// TIA Portal project "学习计数器" (V15.1)

(* hardware
DEVICE "S7-1200 station_1"  S7-1200 Station
   slot 0: "Rack_0"  S7-1200 Rack  Rack  V1.0
   slot 1: "PLC_1"  CPU 1214C DC/DC/DC  6ES7 214-1AG40-0XB0  V4.2
*)

// ===== PLC "PLC_1"  CPU 1214C DC/DC/DC =====

VAR_GLOBAL   // PLC tag table "默认变量表"
   "Tag_1" AT %M0.0 : Bool;
   "Tag_2" AT %M0.1 : Bool;
   "Tag_3" AT %MW100 : Int;
   "Tag_4" AT %Q0.0 : Bool;
   "Tag_5" AT %Q0.1 : Bool;
   "Tag_6" AT %M0.2 : Bool;
   "Tag_7" AT %M0.3 : Bool;
   "Tag_8" AT %MW101 : Int;
   "Tag_9" AT %M0.4 : Bool;
   "Tag_10" AT %M0.5 : Bool;
   "Tag_11" AT %M0.6 : Bool;
   "Tag_12" AT %M0.7 : Bool;
   "Tag_13" AT %MW102 : Int;
   "Tag_14" AT %Q0.2 : Bool;
   "Tag_15" AT %Q0.3 : Bool;
END_VAR

DATA_BLOCK "jishuqi"   // DB4
{ S7_Optimized_Access := 'TRUE' }
VERSION : 0.1
   VAR
      CTU_DB1 : IEC_COUNTER;
   END_VAR
   VAR RETAIN
      CTU_DB2 : IEC_SCOUNTER;
      CTU_DB3 : IEC_DCOUNTER;
      CTD_DB1 : IEC_USCOUNTER;
      CTD_DB2 : IEC_UCOUNTER;
   END_VAR
BEGIN
END_DATA_BLOCK

// folder: System blocks/Program resources

DATA_BLOCK "IEC_Counter_0_DB"   // DB1
{ S7_Optimized_Access := 'TRUE' }
AUTHOR : Simatic
FAMILY : IEC
NAME : CNTR
VERSION : 1.0
// stored: InstanceOfName IEC_COUNTER
"IEC_COUNTER"
BEGIN
END_DATA_BLOCK

DATA_BLOCK "IEC_Counter_0_DB_1"   // DB2
{ S7_Optimized_Access := 'TRUE' }
AUTHOR : Simatic
FAMILY : IEC
NAME : CNTR
VERSION : 1.0
// stored: InstanceOfName IEC_COUNTER
"IEC_COUNTER"
BEGIN
END_DATA_BLOCK

DATA_BLOCK "IEC_Counter_0_DB_2"   // DB3
{ S7_Optimized_Access := 'TRUE' }
AUTHOR : Simatic
FAMILY : IEC
NAME : CNTR
VERSION : 1.0
// stored: InstanceOfName IEC_COUNTER
"IEC_COUNTER"
BEGIN
END_DATA_BLOCK

// folder: (top level)

ORGANIZATION_BLOCK "Main"   // OB1, LAD, ProgramCycle
TITLE = "Main Program Sweep (Cycle)"
{ S7_Optimized_Access := 'TRUE' }
VERSION : 0.1
   VAR_INPUT
      Initial_Call : Bool;   // Initial call of this OB
      Remanence : Bool;   // =True, if remanent data are available
   END_VAR
BEGIN

REGION Network 1: 加计数器
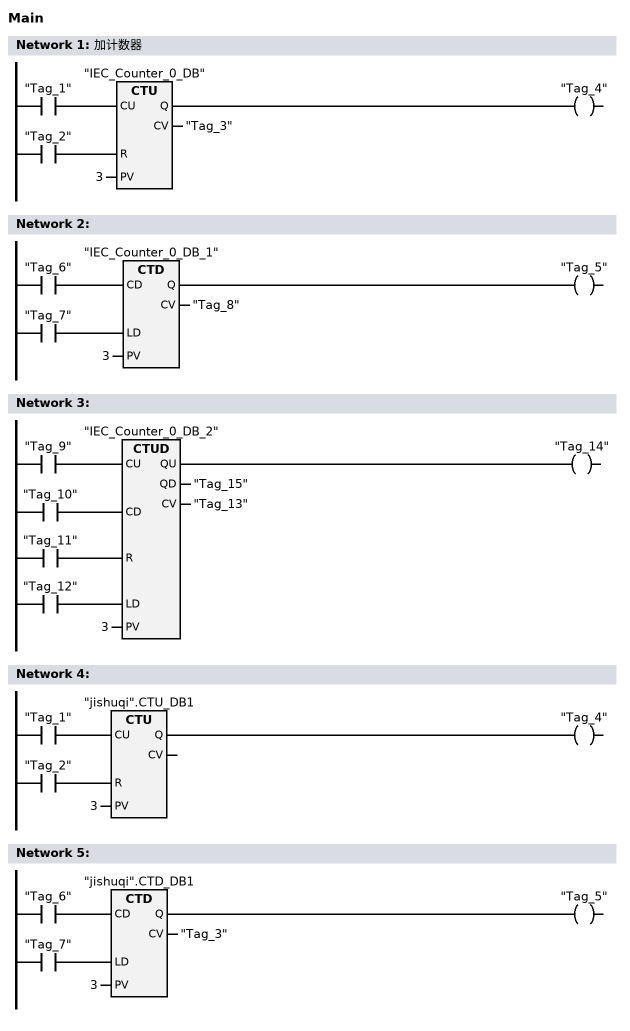
   "IEC_Counter_0_DB".CTU(CU := "Tag_1", R := "Tag_2", PV := 3, CV => "Tag_3");
   "Tag_4" := "IEC_Counter_0_DB".Q;
END_REGION

REGION Network 2
   "IEC_Counter_0_DB_1".CTD(CD := "Tag_6", LD := "Tag_7", PV := 3, CV => "Tag_8");
   "Tag_5" := "IEC_Counter_0_DB_1".Q;
END_REGION

REGION Network 3
   "IEC_Counter_0_DB_2".CTUD(CU := "Tag_9",
                           CD := "Tag_10",
                           R := "Tag_11",
                           LD := "Tag_12",
                           PV := 3,
                           QD => "Tag_15",
                           CV => "Tag_13");
   "Tag_14" := "IEC_Counter_0_DB_2".QU;
END_REGION

REGION Network 4
   "jishuqi".CTU_DB1.CTU(CU := "Tag_1", R := "Tag_2", PV := 3);
   "Tag_4" := "jishuqi".CTU_DB1.Q;
END_REGION

REGION Network 5
   "jishuqi".CTD_DB1.CTD(CD := "Tag_6", LD := "Tag_7", PV := 3, CV => "Tag_3");
   "Tag_5" := "jishuqi".CTD_DB1.Q;
END_REGION
END_ORGANIZATION_BLOCK